// SIMATIC S7-200 project (STEP 7-Micro/WIN), CPU 222 REL 02.01

SYMBOL_TABLE USUARIO1
PARO             I0.0
MARCHA           I0.1
LAMPARA_1        Q0.0
LAMPARA_2        Q0.1
LAMPARA_3        Q0.2
END_SYMBOL_TABLE

ORGANIZATION_BLOCK PRINCIPAL:OB1
TITLE=COMENTARIOS DEL PROGRAMA
BEGIN
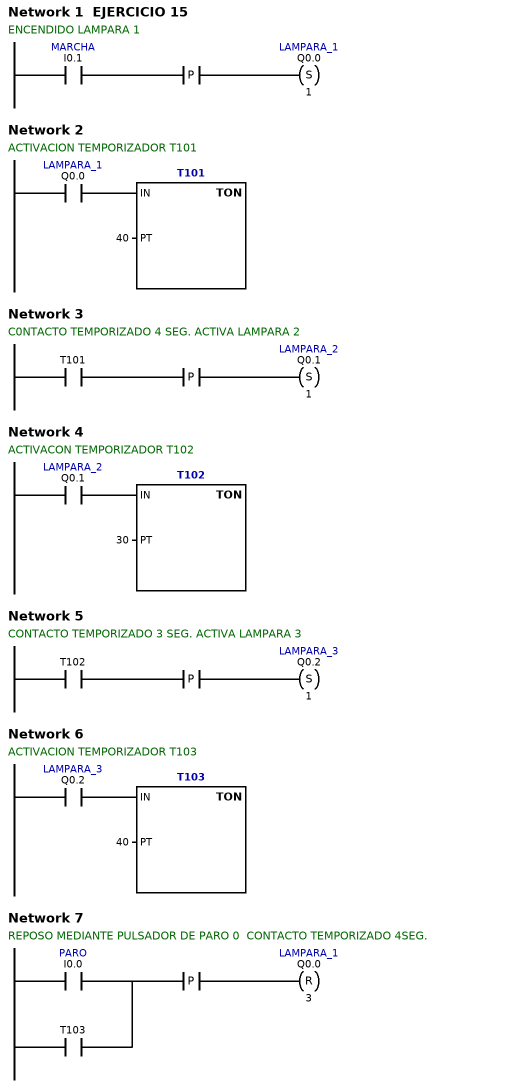
Network 1 // EJERCICIO 15
// ENCENDIDO LAMPARA 1
// (network saved uncompiled; LAD cells follow)
// row 0: c0 -| |- MARCHA:I0.1  c1 -|P|-  c2 -(S) LAMPARA_1:Q0.0, 1
Network 2
// ACTIVACION TEMPORIZADOR T101
// (network saved uncompiled; LAD cells follow)
// row 0: c0 -| |- LAMPARA_1:Q0.0  c1 [TON T101 IN:=power@row0, PT:=40]
// row 1: c1 [box]
Network 3
// C0NTACTO TEMPORIZADO 4 SEG. ACTIVA LAMPARA 2
// (network saved uncompiled; LAD cells follow)
// row 0: c0 -| |- T101  c1 -|P|-  c2 -(S) LAMPARA_2:Q0.1, 1
Network 4
// ACTIVACON TEMPORIZADOR T102
// (network saved uncompiled; LAD cells follow)
// row 0: c0 -| |- LAMPARA_2:Q0.1  c1 [TON T102 IN:=power@row0, PT:=30]
// row 1: c1 [box]
Network 5
// CONTACTO TEMPORIZADO 3 SEG. ACTIVA LAMPARA 3
// (network saved uncompiled; LAD cells follow)
// row 0: c0 -| |- T102  c1 -|P|-  c2 -(S) LAMPARA_3:Q0.2, 1
Network 6
// ACTIVACION TEMPORIZADOR T103
// (network saved uncompiled; LAD cells follow)
// row 0: c0 -| |- LAMPARA_3:Q0.2  c1 [TON T103 IN:=power@row0, PT:=40]
// row 1: c1 [box]
Network 7
// REPOSO MEDIANTE PULSADOR DE PARO 0  CONTACTO TEMPORIZADO 4SEG. 
// (network saved uncompiled; LAD cells follow)
// row 0: c0 -| |- PARO:I0.0 v  c1 -|P|-  c2 -(R) LAMPARA_1:Q0.0, 3
// row 1: c0 -| |- T103 ^
END_ORGANIZATION_BLOCK
